{attribute 'Tc2GvlVarNames'}
{attribute 'pack_mode' := '1'}
VAR_GLOBAL
	
(* ########## Errors ########## *)
	Errors_Cabinet			: TERRORS2;		(* Errors from inside the cabinet *)
	Errors_TwinSAFE			: TERRORS2;		(* TwinSAFE errors *)
	Errors_AutoCycle		: TERRORS2;		(* Errors from the automatic cycles *)
	Errors_Axes				: TERRORS2;		(* Errors from Stober drive axes *)
	Errors_AutoCrossCut		: TERRORS2;		(* Errors Auto CrossCut time out *)
	Errors_LiftingPosition	: TERRORS2;		(* Errors Lifting Position time out *)
	Errors_CrossCutPosition	: TERRORS2;		(* Errors CrossCut Position time out *)
	
(* ########## Warnings ########## *)
	Warnings_Saw			: TERRORS2;		(* Warnings *)

END_VAR

(* stored: Version 1.1.0.1, ProductVersion 3.1.4024.15
   GVL PLCStudio: Id {68d4e592-69bb-456b-bcdd-6a325933713f} *)
